// TIA Portal V15.1 export
// export: Created 2024-06-21T08:41:00.5798838Z, ExportSetting WithDefaults, DisplayName Totally Integrated Automation Portal, DisplayVersion V15.1 Update 5, DisplayName TIA Portal Openness, DisplayVersion V15.1 Update 5, DisplayName SINAMICS Startdrive Advanced, DisplayVersion V15.1, DisplayName G130, G150, S120, S150, SINAMICS MV, S210, DisplayVersion V15.1, DisplayName G110M, G120, G120C, G120D, G120P, DisplayVersion V15.1, DisplayName STEP 7 Professional, DisplayVersion V15.1 Update 5, DisplayName STEP 7 Safety, DisplayVersion V15.1, DisplayName WinCC Professional, DisplayVersion V15.1 Update 5, DisplayName SIMATIC Visualization Architect, DisplayVersion V15.1
FUNCTION_BLOCK "LDBCheck"   // FB2146, FBD
TITLE = LDBCheck
{ S7_Optimized_Access := 'FALSE' }
AUTHOR : VCC
FAMILY : DataHand
VERSION : 0.1
// =============================================================================
// This Module Checks DB Length & DB Number
// =============================================================================
// stored: AutoNumber false, IsIECCheckEnabled true, SetENOAutomatically False, UDAEnableTagReadback false
   VAR_INPUT
      I_DBNr { ExternalAccessible := 'False'; ExternalVisible := 'False'; ExternalWritable := 'False'} : DB_ANY;   // DB
   END_VAR
   VAR_OUTPUT
      O_DBLength { ExternalAccessible := 'False'; ExternalVisible := 'False'; ExternalWritable := 'False'} : Word;   // DB Length
      O_DBNr { ExternalAccessible := 'False'; ExternalVisible := 'False'; ExternalWritable := 'False'} : Word;   // DB Nr
   END_VAR
BEGIN

NETWORK
TITLE = **** 5.2 - Equations - Flow Equations **** Load DB Number & Number
// Load DB Length & Number
      OPN   #I_DBNr;
      L     DBLG;
      T     #O_DBLength;
      L     DBNO;
      T     #O_DBNr;
END_FUNCTION_BLOCK
